Yaskawa INFORM job: BATMAN_4SPOINY2.JBI

/JOB
//NAME BATMAN_4SPOINY2
///FOLDERNAME KRIS-SCIANA
//POS
///NPOS 293,293,243,19,0,0
///TOOL 0
///POSTYPE PULSE
///PULSE
C00000=27461,19727,-15013,5964,93200,7919
C00001=53930,-34836,-43070,10546,92631,-44102
C00002=59372,-32233,-36195,10185,89087,-42536
C00003=59542,-32241,-35992,10174,88938,-42491
C00004=59542,-32142,-35265,10174,88546,-42521
C00005=59542,-32241,-35992,10174,88938,-42491
C00006=60428,-32802,-36126,10115,88624,-42213
C00007=59542,-32241,-35992,10174,88938,-42491
C00008=64039,-48991,-58660,9906,93649,-40580
C00009=69362,-49546,-56329,9460,91325,-38954
C00010=72521,-45533,-52121,9188,90441,-37947
C00011=72521,-45481,-51268,9186,89947,-37982
C00012=72521,-45533,-52121,9188,90441,-37947
C00013=73752,-44607,-51263,9079,90249,-37543
C00014=72521,-45533,-52121,9188,90441,-37947
C00015=72780,-67210,-74355,9190,92926,-37677
C00016=104760,-79002,-75488,1590,83769,10908
C00017=104760,-78316,-71792,1595,81848,10885
C00018=104951,-72146,-66630,1566,81838,10949
C00019=104951,-71977,-65827,1567,81431,10946
C00020=104951,-72146,-66630,1566,81838,10949
C00021=104585,-69689,-65175,1617,82213,10830
C00022=104951,-72146,-66630,1566,81838,10949
C00023=126930,-89810,-77004,-2546,79326,20912
C00024=126930,-86182,-66696,-2587,74851,21005
C00025=124517,-79688,-62407,-2239,75475,20152
C00026=124517,-79372,-61547,-2242,75108,20158
C00027=124517,-79688,-62407,-2239,75475,20152
C00028=123608,-77929,-61403,-2108,75735,19831
C00029=124517,-79688,-62407,-2239,75475,20152
C00030=203387,-120314,-87249,-1260,66339,1853
C00031=200667,-112422,-82916,-708,67693,857
C00032=200667,-111811,-81800,-709,67321,859
C00033=200667,-112422,-82916,-708,67693,857
C00034=202283,-108660,-81695,-1019,68894,1430
C00035=200667,-112422,-82916,-708,67693,857
C00036=197903,-118206,-84689,-161,65798,-138
C00037=190700,-136110,-79236,12987,43309,-5470
C00038=193073,-133711,-78763,11750,43893,-4292
C00039=190700,-136110,-79236,12987,43309,-5470
C00040=190700,-133577,-76218,13120,42767,-5552
C00041=190700,-136110,-79236,12987,43309,-5470
C00042=159264,-85348,-72338,26469,101848,-35770
C00043=164489,-85917,-58916,26689,92487,-35917
C00044=168310,-82776,-58110,27297,92259,-34533
C00045=169943,-81162,-57428,27533,92089,-33955
C00046=168310,-82776,-58110,27297,92259,-34533
C00047=168310,-81475,-55247,27268,91281,-34761
C00048=168310,-82776,-58110,27297,92259,-34533
C00049=174818,-166728,-104111,5010,53468,-9061
C00050=151913,-165072,-108467,9162,58894,-17426
C00051=31054,-58499,-67437,-4813,86361,7552
C00052=17460,-13489,-32841,5083,88285,-10080
C00053=18511,-10450,-28211,4896,86939,-9785
C00054=18511,-10497,-27164,4898,86273,-9811
C00055=18511,-10450,-28211,4896,86939,-9785
C00056=18072,-6386,-24997,4976,87076,-9926
C00057=18511,-10450,-28211,4896,86939,-9785
C00058=19304,-17015,-37138,4755,89006,-9443
C00059=40718,-16031,-27821,-22618,89289,5458
C00060=35897,-12993,-23126,-22071,86757,4185
C00061=35408,-10854,-21474,-22011,86705,4017
C00062=35897,-12993,-23126,-22071,86757,4185
C00063=35897,-12823,-21290,-22084,85788,4364
C00064=35897,-12993,-23126,-22071,86757,4185
C00065=31722,-22647,-27301,-21597,83426,3277
C00066=29589,-18207,-23578,-21312,82862,2603
C00067=29229,-16321,-22176,-21257,82868,2471
C00068=29589,-18207,-23578,-21312,82862,2603
C00069=29589,-17904,-21603,-21354,81873,2778
C00070=29589,-18207,-23578,-21312,82862,2603
C00071=33057,-35215,-50272,-21725,90936,2406
C00072=13245,-10427,-29720,5825,88219,-11479
C00073=13394,-4718,-22818,5800,86900,-11488
C00074=18206,-7497,-25118,4952,86573,-9901
C00075=18519,-8090,-25381,4896,86408,-9803
C00076=21911,-9763,-26755,4284,86207,-8681
C00077=21762,-10624,-27040,4312,85947,-8742
C00078=25203,-13472,-28530,-1187,84834,1033
C00079=19550,-17151,-28181,-117,82684,-851
C00080=19443,-16796,-23929,-6731,81807,11381
C00081=20023,-18123,-24279,-6835,81387,11602
C00082=21850,-21543,-25350,-7161,80456,12281
C00083=15586,-21049,-25758,415,81887,2238
C00084=14598,-19690,-25084,2340,83349,-603
C00085=17410,-32379,-43825,1943,88285,427
C00086=62758,-61083,-67514,9356,96495,3913
C00087=199419,-126821,-93595,-3849,72358,1575
C00088=215588,-96023,-77843,-5493,79414,6921
C00089=206230,-97336,-78342,-4514,78461,3733
C00090=205980,-97628,-78299,-4491,78272,3656
C00091=198784,-97250,-78233,-3683,78060,1181
C00092=198556,-98334,-78334,-3662,77556,1119
C00093=199186,-98644,-78275,-3737,77391,1339
C00094=187587,-121388,-81242,8247,57073,-3790
C00095=198009,-126022,-79257,5356,52636,78
C00096=198735,-126438,-75439,11422,52308,-7805
C00097=182087,-109335,-69935,21135,69891,-28872
C00098=173698,-101527,-65024,22396,76730,-30869
C00099=174667,-108871,-67545,21614,70616,-31488
C00100=190087,-128682,-72511,14911,50768,-12319
C00101=165785,-126013,-84565,21580,74443,-34035
C00102=65346,-79799,-84675,10403,98195,-30166
C00103=73542,-33969,-44608,8971,95126,-24746
C00104=73466,-33578,-44297,8974,95141,-24769
C00105=56512,-3179,-12316,26889,108547,-27571
C00106=55135,-19184,-25463,26231,99696,-30127
C00107=47657,-21774,-22421,25331,99126,-33105
C00108=47657,-23151,-32449,25918,104076,-32001
C00109=58332,-49897,-67983,12473,95404,-30979
C00110=76814,-87681,-77913,12459,85852,-4883
C00111=98077,-64526,-65270,10461,86864,2540
C00112=98077,-64004,-61535,10478,84867,2372
C00113=98452,-64122,-61596,10437,84795,2494
C00114=136766,-62959,-54295,-24287,84543,16325
C00115=133538,-79296,-61255,-19745,72823,18967
C00116=138375,-88192,-61332,-20789,69437,20890
C00117=138917,-90913,-61585,-20643,67750,20404
C00118=142002,-103150,-73880,-19907,68072,18980
C00119=156669,-121711,-96887,-11323,85539,21769
C00120=4467,-137969,-110669,-6539,34039,-3130
C00121=19856,121451,20000,-7167,97699,-79935
C00122=-30106,49565,32966,-7153,97659,-79929
///LIMIT ON
C00123=-48667,-96740,-85237,-4414,71954,-161170
C00124=-50087,-78703,-69642,-4046,71552,-161658
C00125=-49056,-78152,-68509,-4328,71190,-161282
C00126=-50087,-78703,-69642,-4046,71552,-161658
C00127=-51559,-77641,-68057,-3663,71053,-162163
C00128=-50087,-78703,-69642,-4046,71552,-161658
C00129=-68843,-102087,-91870,723,73949,-168126
C00130=-111940,-50657,-63992,-844,88968,-142439
C00131=-116747,-35976,-49037,-28,87281,-144022
C00132=-120801,-38775,-48909,662,85780,-145375
C00133=-120801,-38756,-47729,662,85062,-145378
C00134=-120801,-38775,-48909,662,85780,-145375
C00135=-121754,-36220,-46769,824,85785,-145694
C00136=-120801,-38775,-48909,662,85780,-145375
C00137=-125210,-26619,-58097,1431,97733,-146711
C00138=-131530,-17132,-45035,1132,94544,-146201
C00139=-131530,-17365,-44333,1131,93991,-146205
C00140=-131530,-17132,-45035,1132,94544,-146201
C00141=-132146,-15038,-43228,1237,94517,-146399
C00142=-131530,-17132,-45035,1132,94544,-146201
C00143=-161629,-2767,-38396,12559,109608,-190789
C00144=-160029,-4292,-24208,11904,100070,-191215
C00145=-160029,-4346,-23457,11882,99590,-191262
C00146=-160029,-4292,-24208,11904,100070,-191215
C00147=-159085,-3286,-23121,11882,99786,-190918
C00148=-160029,-4292,-24208,11904,100070,-191215
C00149=-164567,11803,-19941,12295,106250,-192160
C00150=-157312,-13774,-45091,-2984,98065,-146499
C00151=-206670,-20774,-45162,4390,94951,-162466
C00152=-207434,-3536,-26344,4477,92277,-162812
C00153=-207134,-1926,-24499,4435,91966,-162724
C00154=-207434,-3536,-26344,4477,92277,-162812
C00155=-208212,-2907,-24823,4582,91708,-163090
C00156=-207434,-3536,-26344,4477,92277,-162812
C00157=-203791,-18921,-42474,3974,94109,-161555
C00158=-208102,-33336,-45107,4384,70878,-171284
C00159=-208479,-26108,-38450,4536,70518,-171428
C00160=-208501,-36193,-39722,4679,66129,-171606
C00161=-213385,-11527,-27447,11970,86947,-171405
C00162=-211009,-28161,-49573,11590,91579,-170169
C00163=-152191,-54135,-82173,-578,95677,-207495
C00164=-98829,-148789,-110327,23555,60006,-190918
C00165=-63524,-94038,-77380,10109,60123,-176665
C00166=-56536,-89434,-70565,3215,56920,-170295
C00167=-56480,-89635,-70927,3185,57034,-170270
C00168=-58851,-96962,-68332,4510,51796,-171436
C00169=-51054,-86638,-67405,-5688,64202,-168107
C00170=-66960,-121145,-97778,-723,64525,-174040
C00171=-151266,-18842,-50725,13491,96086,-200286
C00172=-151199,-2206,-30574,14854,95015,-197817
C00173=-151558,-2403,-30281,14862,94131,-203931
C00174=-156353,-9182,-30957,16219,92997,-207432
C00175=-161657,-20517,-34126,16277,89446,-208209
C00176=-166380,-28855,-45761,15510,91081,-205955
C00177=-176343,-27519,-58136,14484,97680,-202423
C00178=-146432,-62330,-79152,8575,88774,-157888
C00179=-135076,-29913,-53110,6046,88415,-154204
C00180=-132700,-21303,-45243,5501,87836,-153459
C00181=-120110,-24629,-45165,-11500,84499,-143667
C00182=-116346,-38856,-49381,-12534,80425,-141997
C00183=-112747,-49987,-51295,-13579,76569,-140328
C00184=-112325,-51024,-51497,-13698,76241,-140141
C00185=-106405,-53098,-58914,-14887,80672,-138578
C00186=-95224,-20863,-45190,-12261,93737,-137947
C00187=-95224,-20863,-45190,-12261,93737,-137947
C00188=-95567,-18712,-43618,-12211,93824,-138068
C00189=2669,-23463,-43684,-12198,93814,-143081
C00190=12882,-2853,-23046,-12338,79295,-114850
C00191=140228,6881,-10027,16067,87628,-189683
C00192=178636,-26215,-18003,9541,69682,-178042
C00193=190464,-1998,2686,-1702,78410,-173449
C00194=190464,-1807,3325,-1703,78115,-173446
C00195=190464,-1851,3178,-1703,78183,-173446
C00196=190464,-572,4236,-1705,78187,-173446
C00197=190079,-3448,589,-1660,78950,-173589
C00198=170718,-8896,-1072,11364,69213,-180966
C00199=176690,18547,19438,-1102,83032,-178253
C00200=176690,18907,20631,-1103,82484,-178249
C00201=176690,18865,20492,-1103,82549,-178249
C00202=176937,20672,22196,-1113,82434,-178165
C00203=176690,18518,19335,-1103,83082,-178254
C00204=159096,10761,15360,13640,71000,-185020
C00205=163699,23839,25637,3670,75746,-182781
C00206=163699,24193,26736,3676,75252,-182795
C00207=163699,24137,26562,3674,75330,-182794
C00208=164134,25799,28176,3622,75172,-182647
C00209=163699,23793,25492,3667,75812,-182780
C00210=150784,29671,32882,15137,71440,-188000
C00211=157156,47733,49397,1195,75308,-184939
C00212=157156,48104,50383,1197,74893,-184942
C00213=157156,48016,50149,1197,74991,-184943
C00214=157735,49760,52060,1141,74703,-184746
C00215=157156,47434,48587,1193,75652,-184937
C00216=142367,63352,68521,16801,68626,-191483
C00217=154723,16721,17849,2207,78471,-185762
C00218=154723,17075,19023,2210,77929,-185773
C00219=154723,17004,18788,2210,78036,-185770
C00220=155361,18646,20317,2147,77921,-185553
C00221=154295,15409,15439,2245,79287,-185894
C00222=152548,-46037,-33001,14724,72703,-187200
C00223=173063,-35885,-19745,11040,66557,-180364
C00224=172381,-30459,-14817,12966,67685,-183662
C00225=189647,-41939,-21829,9364,63743,-177626
C00226=212432,-47441,-24871,3550,60965,-169203
C00227=222510,-46248,-24162,762,60877,-165387
C00228=221072,-55571,-31663,-1225,60729,-162686
C00229=183831,-42837,-24403,-640,62781,-163481
C00230=184368,-37494,-19337,-786,62417,-163277
C00231=169590,-25113,-11382,3214,64110,-168775
C00232=153390,312,7747,7325,66459,-174651
C00233=148403,13068,18934,8546,66622,-176472
C00234=147511,16247,21849,8770,66559,-176807
C00235=141966,-23210,-23563,9637,74772,-178174
C00236=49773,-23266,-23600,9630,74761,-174606
C00237=11499,-91272,-60439,14826,66037,-186980
C00238=24614,139305,42242,-12105,94129,-241398
C00239=23281,113263,30549,-9123,91006,-253685
C00240=55336,36118,-12147,-9115,91117,-253682
C00241=110497,-96010,-85203,-9082,91337,-253646
C00242=110132,-97701,-85894,-9078,90857,-326888
C00243=231444,-97696,-85555,14457,66885,-341831
C00244=239081,-48934,-58681,12347,86500,-340546
C00245=232436,-33273,-43061,13430,86148,-342856
C00246=232487,-32587,-41956,13424,85819,-342875
C00247=232487,-32542,-40985,13430,85259,-342937
C00248=232487,-32587,-41956,13424,85819,-342875
C00249=232629,-30129,-40306,13401,86035,-342805
C00250=232487,-32587,-41956,13424,85819,-342875
C00251=213809,-15512,-33444,15950,92576,-348489
C00252=216143,-7692,-23925,15635,90358,-347968
C00253=216143,-7698,-22988,15630,89798,-348040
C00254=216143,-7692,-23925,15635,90358,-347968
C00255=216488,-5395,-22087,15594,90340,-347850
C00256=216143,-7692,-23925,15635,90358,-347968
C00257=207069,12956,-7235,16611,92452,-350833
C00258=206195,16842,-2970,16681,92025,-351195
C00259=206195,16846,-1900,16669,91395,-351281
C00260=206195,16842,-2970,16681,92025,-351195
C00261=206613,19062,-907,16640,91818,-351079
C00262=206195,16842,-2970,16681,92025,-351195
C00263=210833,19416,-576,16221,90958,-349729
C00264=209935,25164,4669,16310,90872,-350053
C00265=209935,25181,5707,16303,90266,-350133
C00266=209935,25164,4669,16310,90872,-350053
C00267=210302,27507,6947,16270,90609,-349961
C00268=209935,25164,4669,16310,90872,-350053
C00269=202776,46738,24588,16950,91193,-352506
C00270=202171,51343,31379,16979,89579,-352941
C00271=202171,51457,32428,16976,89018,-353018
C00272=202171,51343,31379,16979,89579,-352941
C00273=202544,53678,33951,16947,89134,-352871
C00274=202171,51343,31379,16979,89579,-352941
C00275=210768,8740,-16259,16329,94978,-349219
C00276=216926,676,-19392,15562,91669,-347534
C00277=220414,8220,-10388,13170,90389,-353505
C00278=232512,-10946,-26241,11631,88471,-349576
C00279=227494,-25690,-36969,12302,88249,-351307
C00280=237440,-37130,-44669,10939,85718,-348148
C00281=231683,-43662,-56537,11755,90384,-349677
C00282=231683,-43662,-56537,11755,90384,-349677
C00283=240298,-51036,-57572,3930,82785,-334851
C00284=225025,-34742,-47804,6828,86146,-339832
C00285=212279,-13510,-33247,9067,89308,-343887
C00286=207270,-2378,-24690,9890,90330,-345482
C00287=206374,470,-22476,10033,90539,-345765
C00288=201120,-19837,-47084,10933,95828,-347061
C00289=121938,-115164,-95780,1417,89212,-367207
C00290=62315,-114908,-95780,1418,89212,-367206
C00291=62316,-114908,-95779,1418,89212,-367205
C00292=29956,140088,42679,-12136,94183,-404796
///LIMIT OFF
BC00000=80599,337603,478005
BC00001=163893,318206,473102
BC00002=163893,318206,473102
BC00003=163893,318206,473102
BC00004=163893,318206,473102
BC00005=163893,318206,473102
BC00006=163893,318206,473102
BC00007=163893,318206,473102
BC00008=163893,318206,473102
BC00009=163893,318206,473102
BC00010=163893,318206,473102
BC00011=163893,318206,473102
BC00012=163893,318206,473102
BC00013=163893,318206,473102
BC00014=163893,318206,473102
BC00015=163893,318206,473102
BC00016=163893,318206,473102
BC00017=163893,318206,473102
BC00018=163893,318206,473102
BC00019=163893,318206,473102
BC00020=163893,318206,473102
BC00021=163893,318206,473102
BC00022=163893,318206,473102
BC00023=163893,318206,473102
BC00024=163893,318206,473102
BC00025=163893,318206,473102
BC00026=163893,318206,473102
BC00027=163893,318206,473102
BC00028=163893,318206,473102
BC00029=163893,318206,473102
BC00030=163893,318206,473102
BC00031=163893,318206,473102
BC00032=163893,318206,473102
BC00033=163893,318206,473102
BC00034=163893,318206,473102
BC00035=163893,318206,473102
BC00036=163893,318206,473102
BC00037=163893,318206,473102
BC00038=163893,318206,473102
BC00039=163893,318206,473102
BC00040=163893,318206,473102
BC00041=163893,318206,473102
BC00042=163892,318206,473100
BC00043=163892,318207,473095
BC00044=163892,318207,473095
BC00045=163892,318207,473095
BC00046=163892,318207,473095
BC00047=163892,318207,473095
BC00048=163892,318207,473095
BC00049=163893,318206,473102
BC00050=163893,318206,473102
BC00051=163893,318206,473102
BC00052=163893,318206,473102
BC00053=163893,318206,473102
BC00054=163893,318206,473102
BC00055=163893,318206,473102
BC00056=163893,318206,473102
BC00057=163893,318206,473102
BC00058=163893,318206,473102
BC00059=163893,318206,473102
BC00060=163893,318206,473102
BC00061=163893,318206,473102
BC00062=163893,318206,473102
BC00063=163893,318206,473102
BC00064=163893,318206,473102
BC00065=163893,318206,473102
BC00066=163893,318206,473102
BC00067=163893,318206,473102
BC00068=163893,318206,473102
BC00069=163893,318206,473102
BC00070=163893,318206,473102
BC00071=163893,318206,473102
BC00072=163893,318206,473102
BC00073=163893,318206,473102
BC00074=163893,318206,473102
BC00075=163893,318206,473102
BC00076=163893,318206,473102
BC00077=163893,318206,473102
BC00078=163893,318206,473102
BC00079=163893,318206,473102
BC00080=163893,318206,473102
BC00081=163893,318206,473102
BC00082=163893,318206,473102
BC00083=163894,318206,473105
BC00084=163894,318206,473105
BC00085=163894,318206,473105
BC00086=163894,318207,608827
BC00087=163894,318207,473102
BC00088=163894,318207,473102
BC00089=163894,318207,473102
BC00090=163894,318207,473102
BC00091=163894,318207,473102
BC00092=163894,318207,473102
BC00093=163894,318207,473102
BC00094=163894,318207,473102
BC00095=163894,318207,473102
BC00096=163894,318207,473102
BC00097=163894,318207,473102
BC00098=163894,318207,473102
BC00099=163894,318207,473102
BC00100=163894,318207,473102
BC00101=163894,318207,473102
BC00102=163894,318207,473102
BC00103=163894,318207,473102
BC00104=163894,318207,473102
BC00105=163894,318207,473102
BC00106=163894,318207,473102
BC00107=163894,318207,473102
BC00108=163894,318207,473102
BC00109=163894,318207,473102
BC00110=163894,318207,473102
BC00111=163894,318207,473102
BC00112=163894,318207,473102
BC00113=163894,318207,473102
BC00114=163894,318207,473102
BC00115=163894,318207,473102
BC00116=163894,318207,473102
BC00117=163894,318207,473102
BC00118=163894,318207,473102
BC00119=163894,318207,706181
BC00120=112319,5379,1050005
BC00121=125260,5957,1075157
BC00122=125260,5957,1075157
BC00123=255263,5047,617472
BC00124=255263,5047,617472
BC00125=255263,5047,617472
BC00126=255263,5047,617472
BC00127=255263,5047,617472
BC00128=255263,5047,617472
BC00129=255263,5047,617472
BC00130=255263,5047,617472
BC00131=255263,5047,617472
BC00132=255263,5047,617472
BC00133=255263,5047,617472
BC00134=255263,5047,617472
BC00135=255263,5047,617472
BC00136=255263,5047,617472
BC00137=255263,5047,617472
BC00138=255263,5047,617472
BC00139=255263,5047,617472
BC00140=255263,5047,617472
BC00141=255263,5047,617472
BC00142=255263,5047,617472
BC00143=255263,5047,617472
BC00144=255263,5047,617472
BC00145=255263,5047,617472
BC00146=255263,5047,617472
BC00147=255263,5047,617472
BC00148=255263,5047,617472
BC00149=255263,5047,617472
BC00150=255263,5047,617472
BC00151=255263,5047,617472
BC00152=255263,5047,617472
BC00153=255262,5048,617469
BC00154=255263,5047,617472
BC00155=255263,5047,617472
BC00156=255263,5047,617472
BC00157=255263,5047,617472
BC00158=255263,5047,617472
BC00159=255263,5047,617472
BC00160=255263,5047,617472
BC00161=255263,5047,617472
BC00162=255263,5047,617472
BC00163=255262,5047,617469
BC00164=255262,5047,617469
BC00165=255262,5047,617469
BC00166=255262,5047,617469
BC00167=255261,5048,617462
BC00168=255261,5048,617462
BC00169=255261,5048,617462
BC00170=255261,5048,617462
BC00171=255261,5048,617462
BC00172=255261,5048,617460
BC00173=255261,5048,617460
BC00174=255261,5048,617460
BC00175=255261,5048,617460
BC00176=255261,5048,617460
BC00177=255261,5048,617460
BC00178=255261,5048,617460
BC00179=255262,5048,617458
BC00180=255262,5048,617458
BC00181=255262,5048,617458
BC00182=255262,5048,617458
BC00183=255262,5048,617458
BC00184=255262,5048,617458
BC00185=255262,5048,617458
BC00186=255262,5048,1054021
BC00187=364357,5048,1054021
BC00188=346085,493744,1054021
BC00189=119927,493744,1054021
BC00190=122126,493982,1062735
BC00191=316085,494322,354264
BC00192=316085,376158,354264
BC00193=316085,376158,354264
BC00194=316085,376158,354264
BC00195=316085,376158,354264
BC00196=316085,376158,354264
BC00197=316085,376158,354264
BC00198=316085,376158,354264
BC00199=316085,376158,354264
BC00200=316085,376158,354264
BC00201=316085,376158,354264
BC00202=316085,376158,354264
BC00203=316085,376158,354264
BC00204=316085,376158,354264
BC00205=316085,376158,354264
BC00206=316085,376158,354264
BC00207=316085,376158,354264
BC00208=316085,376158,354264
BC00209=316085,376158,354264
BC00210=316085,376158,354264
BC00211=316085,376158,354264
BC00212=316085,376158,354264
BC00213=316085,376158,354264
BC00214=316085,376158,354264
BC00215=316085,376158,354264
BC00216=316085,376158,354264
BC00217=316085,310375,354264
BC00218=316085,310375,354264
BC00219=316085,310375,354264
BC00220=316085,310375,354264
BC00221=316085,310375,354264
BC00222=316085,310375,354264
BC00223=316085,310375,354264
BC00224=316083,310375,354262
BC00225=316083,310375,354262
BC00226=316083,310375,354262
BC00227=316083,310375,354262
BC00228=316083,310375,354262
BC00229=316083,310375,354262
BC00230=316083,310375,354262
BC00231=316083,310375,354262
BC00232=316083,310375,354262
BC00233=316083,310375,354262
BC00234=316083,310375,354262
BC00235=316083,310374,354261
BC00236=221693,504700,545055
BC00237=139211,579237,982811
BC00238=124231,580310,1074882
BC00239=85429,579747,1064499
BC00240=244755,514688,1010883
BC00241=393595,402951,918797
BC00242=393595,99043,918797
BC00243=393595,99043,199678
BC00244=398179,136533,199678
BC00245=398179,136533,199674
BC00246=398179,136533,199674
BC00247=398179,136533,199674
BC00248=398179,136533,199674
BC00249=398179,136533,199674
BC00250=398179,136533,199674
BC00251=398179,136533,199674
BC00252=398179,136532,199672
BC00253=398179,136532,199672
BC00254=398179,136532,199672
BC00255=398179,136532,199672
BC00256=398179,136532,199672
BC00257=398179,136532,199672
BC00258=398179,136532,199672
BC00259=398179,136532,199672
BC00260=398179,136532,199672
BC00261=398179,136532,199672
BC00262=398179,136532,199672
BC00263=398179,99664,199672
BC00264=398179,99664,199672
BC00265=398179,99664,199672
BC00266=398179,99664,199672
BC00267=398179,99664,199672
BC00268=398179,99664,199672
BC00269=398179,99664,199672
BC00270=398179,99664,199672
BC00271=398179,99664,199672
BC00272=398179,99664,199672
BC00273=398179,99664,199672
BC00274=398179,99664,199672
BC00275=398179,99664,199672
BC00276=398179,99664,199672
BC00277=398179,99664,199672
BC00278=398179,99664,199672
BC00279=398179,149360,199672
BC00280=398179,149360,199672
BC00281=398179,149360,199672
BC00282=351196,62906,171676
BC00283=351196,62906,171676
BC00284=351196,62906,171676
BC00285=351196,62906,171676
BC00286=351196,62906,171676
BC00287=351196,62906,171676
BC00288=351196,62906,171676
BC00289=397107,62906,780423
BC00290=397107,492277,780423
BC00291=397107,492277,780421
BC00292=68537,642032,1075143
EC00000=-811452,-554689
EC00001=-811450,-554689
EC00002=-811450,-554689
EC00003=-811450,-554689
EC00004=-811450,-554689
EC00005=-811450,-554689
EC00006=-811450,-554689
EC00007=-811450,-554689
EC00008=-811450,-554689
EC00009=-811450,-554689
EC00010=-811450,-554689
EC00011=-811450,-554689
EC00012=-811450,-554689
EC00013=-811450,-554689
EC00014=-811450,-554689
EC00015=-811450,-554689
EC00016=-811450,-554689
EC00017=-811450,-554689
EC00018=-811450,-554689
EC00019=-811450,-554689
EC00020=-811450,-554689
EC00021=-811450,-554689
EC00022=-811450,-554689
EC00023=-811450,-554689
EC00024=-811450,-554689
EC00025=-811450,-554689
EC00026=-811450,-554689
EC00027=-811450,-554689
EC00028=-811450,-554689
EC00029=-811450,-554689
EC00030=-811447,-554690
EC00031=-811443,-554690
EC00032=-811443,-554690
EC00033=-811443,-554690
EC00034=-811443,-554690
EC00035=-811450,-554689
EC00036=-811450,-554689
EC00037=-811450,-554689
EC00038=-811450,-554689
EC00039=-811450,-554689
EC00040=-811450,-554689
EC00041=-811450,-554689
EC00042=-811450,-554689
EC00043=-811450,-554689
EC00044=-811450,-554689
EC00045=-811450,-554689
EC00046=-811450,-554689
EC00047=-811450,-554689
EC00048=-811450,-554689
EC00049=-811450,-554689
EC00050=-811450,-554689
EC00051=-811450,-554689
EC00052=-811450,-554689
EC00053=-811450,-554689
EC00054=-811450,-554689
EC00055=-811450,-554689
EC00056=-811450,-554689
EC00057=-811450,-554689
EC00058=-811450,-554689
EC00059=-811450,-554689
EC00060=-811450,-554689
EC00061=-811450,-554689
EC00062=-811450,-554689
EC00063=-811452,-554689
EC00064=-811452,-554689
EC00065=-811452,-554689
EC00066=-811451,-554689
EC00067=-811451,-554689
EC00068=-811451,-554689
EC00069=-811451,-554689
EC00070=-811451,-554689
EC00071=-811451,-554689
EC00072=-811451,-554689
EC00073=-811451,-554689
EC00074=-811451,-554689
EC00075=-811451,-554689
EC00076=-811451,-554689
EC00077=-811451,-554689
EC00078=-811451,-554689
EC00079=-811451,-554689
EC00080=-811451,-554689
EC00081=-811451,-554689
EC00082=-811451,-554689
EC00083=-811451,-554689
EC00084=-811451,-554689
EC00085=-811451,-554689
EC00086=-811451,-554689
EC00087=-811451,-554689
EC00088=-811451,-554689
EC00089=-811451,-554689
EC00090=-811451,-554689
EC00091=-811451,-554689
EC00092=-811451,-554689
EC00093=-811451,-554689
EC00094=-811451,-554689
EC00095=-811451,-554689
EC00096=-811451,-554689
EC00097=-811451,-554689
EC00098=-811451,-554689
EC00099=-811451,-554689
EC00100=-363208,-550746
EC00101=-363208,-550746
EC00102=-363208,-550746
EC00103=-363208,-550746
EC00104=-363208,-550746
EC00105=-363208,-550746
EC00106=-363208,-550746
EC00107=-363208,-550746
EC00108=-363208,-550746
EC00109=-363208,-550746
EC00110=-363208,-550746
EC00111=-363208,-550746
EC00112=-363208,-550746
EC00113=-363208,-550746
EC00114=-363208,-550746
EC00115=-363208,-550746
EC00116=-363208,-550746
EC00117=-363208,-550746
EC00118=-363208,-550746
EC00119=-363208,-550746
EC00120=-363208,-550746
EC00121=-363208,-550746
EC00122=-363208,-550746
EC00123=-363208,-550746
EC00124=-363208,-550746
EC00125=-363208,-550746
EC00126=-363208,-550746
EC00127=-363208,-550746
EC00128=-363208,-550746
EC00129=-363208,-550746
EC00130=-363208,-550746
EC00131=-363208,-550746
EC00132=-363208,-550746
EC00133=-363208,-550746
EC00134=-363208,-550746
EC00135=-363208,-550746
EC00136=-363208,-550746
EC00137=-363207,-550746
EC00138=-363207,-550746
EC00139=-363207,-550746
EC00140=-363207,-550746
EC00141=-363207,-550746
EC00142=-363206,-550746
EC00143=-363206,-550746
EC00144=-363206,-550746
EC00145=-363206,-550746
EC00146=-363206,-550746
EC00147=-363206,-550746
EC00148=-363206,-550746
EC00149=-363206,-550746
EC00150=-363206,-550746
EC00151=-363206,-550746
EC00152=-363206,-550746
EC00153=-363206,-550746
EC00154=-363206,-550746
EC00155=-363206,-550746
EC00156=-363206,-550746
EC00157=-363206,-550746
EC00158=0,0
EC00159=-802750,0
EC00160=-802750,0
EC00161=-802750,0
EC00162=-802750,0
EC00163=-802750,0
EC00164=-802750,0
EC00165=-802750,0
EC00166=-802750,0
EC00167=-802750,0
EC00168=-802750,0
EC00169=-802750,0
EC00170=-802750,0
EC00171=-802750,0
EC00172=-802750,0
EC00173=-802750,0
EC00174=-802750,0
EC00175=-802750,0
EC00176=-802750,0
EC00177=-802750,0
EC00178=-802750,0
EC00179=-802750,0
EC00180=-802750,0
EC00181=-802750,0
EC00182=-802750,0
EC00183=-802750,0
EC00184=-802749,0
EC00185=-802749,0
EC00186=-802749,0
EC00187=-802749,0
EC00188=-802749,0
EC00189=-802749,0
EC00190=-802749,0
EC00191=-802749,0
EC00192=-802749,0
EC00193=-802749,0
EC00194=-802749,0
EC00195=-802748,0
EC00196=-802748,0
EC00197=793507,0
EC00198=793506,-1
EC00199=793506,-1
EC00200=793506,-1
EC00201=793506,-1
EC00202=793506,-1
EC00203=793506,-1
EC00204=793506,-1
EC00205=793505,-1
EC00206=793505,-1
EC00207=793505,-1
EC00208=793505,-1
EC00209=793505,-1
EC00210=793504,-1
EC00211=793504,-1
EC00212=793504,-1
EC00213=793504,-1
EC00214=793504,-1
EC00215=793504,-1
EC00216=793504,-1
EC00217=793504,-1
EC00218=793504,-1
EC00219=793504,-1
EC00220=793504,-1
EC00221=793504,-1
EC00222=793504,-1
EC00223=793504,-1
EC00224=793504,-1
EC00225=793504,-1
EC00226=793504,-1
EC00227=793504,-1
EC00228=793504,-1
EC00229=793504,-1
EC00230=793504,-1
EC00231=793504,-1
EC00232=793504,-1
EC00233=793504,-1
EC00234=793504,-1
EC00235=793504,-1
EC00236=793504,-1
EC00237=793504,-1
EC00238=793504,-1
EC00239=793504,-1
EC00240=793504,-1
EC00241=793503,548424
EC00242=0,-1
///POSTYPE BASE
///RECTAN
///RCONF 0,0,0,0,1,0,0,0,0,0,0,0,0,0,0,0,0,0,0,0,0,0,0,0
P00006=2.006,1.622,-0.565,0.0000,0.0000,0.0000
P00021=0.073,2.058,-0.109,0.0000,0.0000,0.0000
P00022=2.006,1.622,-0.565,0.0000,0.0000,0.0000
///RCONF 0,0,0,0,0,0,0,0,0,0,0,0,0,0,0,0,0,0,0,0,0,0,0,0
P00023=-2.957,-4.083,2.762,0.0000,0.0000,0.0000
P00024=-1.466,-0.226,-0.419,0.0000,0.0000,0.0000
P00025=3.643,0.007,-2.585,0.0000,0.0000,0.0000
P00026=2.644,0.055,-2.583,0.0000,0.0000,0.0000
P00027=2.278,0.099,-4.210,0.0000,0.0000,0.0000
P00028=-1.778,-0.182,-2.050,0.0000,0.0000,0.0000
P00029=1.749,4.006,-0.261,0.0000,0.0000,0.0000
P00030=-0.014,-0.768,0.131,0.0000,0.0000,0.0000
///RCONF 0,0,0,0,1,0,0,0,0,0,0,0,0,0,0,0,0,0,0,0,0,0,0,0
P00034=-8.151,9.743,-4.393,0.0000,0.0000,0.0000
///RCONF 0,0,0,0,0,0,0,0,0,0,0,0,0,0,0,0,0,0,0,0,0,0,0,0
P00035=0.390,-0.027,1.040,0.0000,0.0000,0.0000
P00036=-2.434,0.084,0.197,0.0000,0.0000,0.0000
P00037=-1.075,5.090,-3.949,0.0000,0.0000,0.0000
P00040=2.716,-0.016,3.014,0.0000,0.0000,0.0000
P00041=-0.109,0.014,0.966,0.0000,0.0000,0.0000
P00042=-0.220,0.371,-0.613,0.0000,0.0000,0.0000
P00043=-0.179,-5.890,-3.227,0.0000,0.0000,0.0000
//INST
///DATE 2024/07/30 17:33
///ATTR SC,RW
///GROUP1 RB1,BS1
///GROUP2 ST1
NOP
SFTOF
MOVJ C00000 BC00000 VJ=100.00  +MOVJ EC00000 VJ=100.00
'SZUKANIE
SFTOF
MOVJ C00001 BC00001 VJ=100.00  +MOVJ EC00001 VJ=30.00
MOVL C00002 BC00002 V=83.3  +MOVJ EC00002 VJ=15.00
MOVL C00003 BC00003 V=83.3  +MOVJ EC00003 VJ=15.00
REFP 3 RB1 C00004 BC00004
CALL JOB:SEARCH-R1
SET P026 P006
SFTON P026
MOVL C00005 BC00005 V=83.3  +MOVJ EC00004 VJ=15.00
REFP 3 RB1 C00006 BC00006
CALL JOB:SEARCH-R1
SET P026 P006
MOVL C00007 BC00007 V=83.3  +MOVJ EC00005 VJ=15.00
SFTOF
MOVL C00008 BC00008 V=83.3  +MOVJ EC00006 VJ=15.00
MOVL C00009 BC00009 V=83.3  +MOVJ EC00007 VJ=15.00
MOVL C00010 BC00010 V=83.3  +MOVJ EC00008 VJ=15.00
REFP 3 RB1 C00011 BC00011
CALL JOB:SEARCH-R1
SET P027 P006
SFTON P027
MOVL C00012 BC00012 V=83.3  +MOVJ EC00009 VJ=15.00
REFP 3 RB1 C00013 BC00013
CALL JOB:SEARCH-R1
SET P027 P006
MOVL C00014 BC00014 V=83.3  +MOVJ EC00010 VJ=15.00
SFTOF
MOVJ C00015 BC00015 VJ=100.00  +MOVJ EC00011 VJ=100.00
SFTOF
MOVJ C00016 BC00016 VJ=100.00  +MOVJ EC00012 VJ=100.00
MOVL C00017 BC00017 V=83.3  +MOVJ EC00013 VJ=15.00
MOVL C00018 BC00018 V=83.3  +MOVJ EC00014 VJ=15.00
REFP 3 RB1 C00019 BC00019
CALL JOB:SEARCH-R1
SET P029 P006
SFTON P029
MOVL C00020 BC00020 V=83.3  +MOVJ EC00015 VJ=15.00
REFP 3 RB1 C00021 BC00021
CALL JOB:SEARCH-R1
SET P029 P006
MOVL C00022 BC00022 V=83.3  +MOVJ EC00016 VJ=15.00
SFTOF
MOVL C00023 BC00023 V=83.3  +MOVJ EC00017 VJ=15.00
MOVL C00024 BC00024 V=83.3  +MOVJ EC00018 VJ=15.00
MOVL C00025 BC00025 V=83.3  +MOVJ EC00019 VJ=15.00
REFP 3 RB1 C00026 BC00026
CALL JOB:SEARCH-R1
SET P030 P006
SFTON P030
MOVL C00027 BC00027 V=83.3  +MOVJ EC00020 VJ=15.00
REFP 3 RB1 C00028 BC00028
CALL JOB:SEARCH-R1
SET P030 P006
MOVL C00029 BC00029 V=83.3  +MOVJ EC00021 VJ=15.00
SFTOF
MOVL C00030 BC00030 V=250.0  +MOVJ EC00022 VJ=15.00
MOVL C00031 BC00031 V=83.3  +MOVJ EC00023 VJ=15.00
REFP 3 RB1 C00032 BC00032
CALL JOB:SEARCH-R1
SET P036 P006
SFTON P036
MOVL C00033 BC00033 V=83.3  +MOVJ EC00024 VJ=15.00
REFP 3 RB1 C00034 BC00034
CALL JOB:SEARCH-R1
SET P036 P006
MOVL C00035 BC00035 V=83.3  +MOVJ EC00025 VJ=15.00
SFTOF
MOVL C00036 BC00036 V=11.0  +MOVJ EC00026 VJ=0.78
MOVL C00037 BC00037 V=83.3  +MOVJ EC00027 VJ=15.00
REFP 3 RB1 C00038 BC00038
CALL JOB:SEARCH-R1
SET P040 P006
SFTON P040
MOVL C00039 BC00039 V=83.3  +MOVJ EC00028 VJ=15.00
REFP 3 RB1 C00040 BC00040
CALL JOB:SEARCH-R1
SET P040 P006
MOVL C00041 BC00041 V=83.3  +MOVJ EC00029 VJ=15.00
SFTOF
MOVJ C00042 BC00042 VJ=100.00  +MOVJ EC00030 VJ=0.78
MOVJ C00043 BC00043 VJ=100.00  +MOVJ EC00031 VJ=100.00
MOVL C00044 BC00044 V=83.3  +MOVJ EC00032 VJ=15.00
REFP 3 RB1 C00045 BC00045
CALL JOB:SEARCH-R1
SET P041 P006
SFTON P041
MOVL C00046 BC00046 V=83.3  +MOVJ EC00033 VJ=15.00
REFP 3 RB1 C00047 BC00047
CALL JOB:SEARCH-R1
SET P041 P006
MOVL C00048 BC00048 V=83.3  +MOVJ EC00034 VJ=15.00
SFTOF
MOVL C00049 BC00049 V=250.0  +MOVJ EC00035 VJ=15.00
MOVJ C00050 BC00050 VJ=100.00  +MOVJ EC00036 VJ=15.00
MOVJ C00051 BC00051 VJ=100.00  +MOVJ EC00037 VJ=100.00
MOVJ C00052 BC00052 VJ=100.00  +MOVJ EC00038 VJ=100.00
MOVL C00053 BC00053 V=83.3  +MOVJ EC00039 VJ=15.00
REFP 3 RB1 C00054 BC00054
CALL JOB:SEARCH-R1
SET P037 P006
SFTON P037
MOVL C00055 BC00055 V=83.3  +MOVJ EC00040 VJ=15.00
REFP 3 RB1 C00056 BC00056
CALL JOB:SEARCH-R1
SET P037 P006
MOVL C00057 BC00057 V=83.3  +MOVJ EC00041 VJ=15.00
MOVJ C00058 BC00058 VJ=100.00  +MOVJ EC00042 VJ=100.00
MOVJ C00059 BC00059 VJ=100.00  +MOVJ EC00043 VJ=100.00
MOVL C00060 BC00060 V=83.3  +MOVJ EC00044 VJ=15.00
REFP 3 RB1 C00061 BC00061
CALL JOB:SEARCH-R1
SET P042 P006
SFTOF
SFTON P042
MOVL C00062 BC00062 V=83.3  +MOVJ EC00045 VJ=15.00
REFP 3 RB1 C00063 BC00063
CALL JOB:SEARCH-R1
SET P042 P006
MOVL C00064 BC00064 V=83.3  +MOVJ EC00046 VJ=15.00
SFTOF
MOVJ C00065 BC00065 VJ=100.00  +MOVJ EC00047 VJ=100.00
MOVL C00066 BC00066 V=83.3  +MOVJ EC00048 VJ=15.00
REFP 3 RB1 C00067 BC00067
CALL JOB:SEARCH-R1
SET P042 P006
SFTON P042
MOVL C00068 BC00068 V=83.3  +MOVJ EC00049 VJ=15.00
REFP 3 RB1 C00069 BC00069
CALL JOB:SEARCH-R1
SET P042 P006
MOVL C00070 BC00070 V=83.3  +MOVJ EC00050 VJ=15.00
SFTOF
MOVJ C00071 BC00071 VJ=100.00  +MOVJ EC00051 VJ=100.00
SFTOF
MOVL C00072 BC00072 V=166.7  +MOVJ EC00052 VJ=15.00
SFTON P037
MACRO1 MJ#(0) ARGF7
MOVL C00073 BC00073 V=83.3  +MOVJ EC00053 VJ=100.00
ARCON
MOVL C00074 BC00074 V=10.0  +MOVJ EC00054 VJ=100.00
MOVL C00075 BC00075 V=10.0  +MOVJ EC00055 VJ=100.00
MOVL C00076 BC00076 V=10.0  +MOVJ EC00056 VJ=100.00
MOVL C00077 BC00077 V=10.0  +MOVJ EC00057 VJ=100.00
MOVL C00078 BC00078 V=10.0  +MOVJ EC00058 VJ=100.00
SFTOF
SFTON P042
MOVL C00079 BC00079 V=10.0  +MOVJ EC00059 VJ=100.00
SFTOF
SFTON P043
MOVL C00080 BC00080 V=10.0  +MOVJ EC00060 VJ=100.00
MACRO1 MJ#(0) ARGF7
MOVL C00081 BC00081 V=10.0  +MOVJ EC00061 VJ=100.00
MOVL C00082 BC00082 V=10.0  +MOVJ EC00062 VJ=100.00
MOVL C00083 BC00083 V=10.0  +MOVJ EC00063 VJ=100.00
MOVL C00084 BC00084 V=10.0  +MOVJ EC00064 VJ=20.00
ARCOF
MOVJ C00085 BC00085 VJ=20.00  +MOVJ EC00065 VJ=20.00
SFTOF
MOVJ C00086 BC00086 VJ=100.00  +MOVJ EC00066 VJ=20.00
MOVJ C00087 BC00087 VJ=100.00  +MOVJ EC00067 VJ=20.00
SFTON P036
MOVJ C00088 BC00088 VJ=20.00  +MOVJ EC00068 VJ=100.00
ARCON
MOVL C00089 BC00089 V=10.0  +MOVJ EC00069 VJ=20.00
TIMER T=0.10
MOVL C00090 BC00090 V=8.3  +MOVJ EC00070 VJ=20.00
MOVL C00091 BC00091 V=8.3  +MOVJ EC00071 VJ=20.00
MOVL C00092 BC00092 V=10.0  +MOVJ EC00072 VJ=20.00
MOVL C00093 BC00093 V=10.0  +MOVJ EC00073 VJ=20.00
MOVL C00094 BC00094 V=10.0  +MOVJ EC00074 VJ=20.00
SFTOF
SFTON P040
MOVL C00095 BC00095 V=10.0  +MOVJ EC00075 VJ=20.00
MOVL C00096 BC00096 V=10.0  +MOVJ EC00076 VJ=20.00
SFTOF
SFTON P041
MOVL C00097 BC00097 V=10.0  +MOVJ EC00077 VJ=20.00
ARCON
MOVL C00098 BC00098 V=10.0  +MOVJ EC00078 VJ=20.00
MOVL C00099 BC00099 V=10.0  +MOVJ EC00079 VJ=50.00
MOVL C00100 BC00100 V=10.0  +MOVJ EC00080 VJ=15.00
ARCOF
MOVJ C00101 BC00101 VJ=15.00  +MOVJ EC00081 VJ=15.00
SFTOF
MOVJ C00102 BC00102 VJ=30.00  +MOVJ EC00082 VJ=30.00
SFTON P027
MOVJ C00103 BC00103 VJ=30.00  +MOVJ EC00083 VJ=30.00
ARCON
MOVL C00104 BC00104 V=10.0  +MOVJ EC00084 VJ=100.00
MOVL C00105 BC00105 V=10.0  +MOVJ EC00085 VJ=20.00
SFTOF
SFTON P026
MOVL C00106 BC00106 V=10.0  +MOVJ EC00086 VJ=20.00
MOVL C00107 BC00107 V=10.0  +MOVJ EC00087 VJ=20.00
ARCOF
SFTOF
MOVJ C00108 BC00108 VJ=100.00  +MOVJ EC00088 VJ=20.00
MOVJ C00109 BC00109 VJ=30.00  +MOVJ EC00089 VJ=30.00
MOVJ C00110 BC00110 VJ=100.00  +MOVJ EC00090 VJ=20.00
MOVJ C00111 BC00111 VJ=30.00  +MOVJ EC00091 VJ=30.00
SFTON P029
MOVJ C00112 BC00112 VJ=30.00  +MOVJ EC00092 VJ=30.00
ARCON
MOVL C00113 BC00113 V=10.0  +MOVJ EC00093 VJ=20.00
MOVL C00114 BC00114 V=10.0  +MOVJ EC00094 VJ=20.00
SFTOF
SFTON P030
MOVL C00115 BC00115 V=10.0  +MOVJ EC00095 VJ=20.00
MOVL C00116 BC00116 V=10.0  +MOVJ EC00096 VJ=20.00
MOVL C00117 BC00117 V=10.0  +MOVJ EC00097 VJ=20.00
ARCOF
MOVJ C00118 BC00118 VJ=20.00  +MOVJ EC00098 VJ=20.00
SFTOF
MOVJ C00119 BC00119 VJ=100.00  +MOVJ EC00099 VJ=100.00
MOVJ C00120 BC00120 VJ=100.00  +MOVJ EC00100 VJ=100.00
CALL JOB:CLEAN-R1_LONG
MOVJ C00121 BC00121 VJ=100.00  +MOVJ EC00101 VJ=100.00
MOVJ C00122 BC00122 VJ=100.00  +MOVJ EC00102 VJ=100.00
'SZUKANIE DRUGA STRONA
MOVJ C00123 BC00123 VJ=30.00  +MOVJ EC00103 VJ=15.00
SFTOF
MOVL C00124 BC00124 V=83.3  +MOVJ EC00104 VJ=15.00
REFP 3 RB1 C00125 BC00125
CALL JOB:SEARCH-R1
SET P035 P006
SFTON P035
MOVL C00126 BC00126 V=83.3  +MOVJ EC00105 VJ=15.00
REFP 3 RB1 C00127 BC00127
CALL JOB:SEARCH-R1
SET P035 P006
MOVL C00128 BC00128 V=83.3  +MOVJ EC00106 VJ=15.00
SFTOF
MOVJ C00129 BC00129 VJ=50.00  +MOVJ EC00107 VJ=50.00
MOVJ C00130 BC00130 VJ=15.00  +MOVJ EC00108 VJ=15.00
MOVL C00131 BC00131 V=83.3  +MOVJ EC00109 VJ=15.00
MOVL C00132 BC00132 V=83.3  +MOVJ EC00110 VJ=15.00
REFP 3 RB1 C00133 BC00133
CALL JOB:SEARCH-R1
SET P026 P006
SFTON P026
MOVL C00134 BC00134 V=83.3  +MOVJ EC00111 VJ=15.00
REFP 3 RB1 C00135 BC00135
CALL JOB:SEARCH-R1
SET P026 P006
MOVL C00136 BC00136 V=83.3  +MOVJ EC00112 VJ=15.00
SFTOF
MOVL C00137 BC00137 V=83.3  +MOVJ EC00113 VJ=15.00
MOVL C00138 BC00138 V=83.3  +MOVJ EC00114 VJ=15.00
REFP 3 RB1 C00139 BC00139
CALL JOB:SEARCH-R1
SET P027 P006
SFTON P027
MOVL C00140 BC00140 V=83.3  +MOVJ EC00115 VJ=15.00
REFP 3 RB1 C00141 BC00141
CALL JOB:SEARCH-R1
SET P027 P006
MOVL C00142 BC00142 V=83.3  +MOVJ EC00116 VJ=15.00
SFTOF
MOVL C00143 BC00143 V=83.3  +MOVJ EC00117 VJ=15.00
MOVL C00144 BC00144 V=83.3  +MOVJ EC00118 VJ=15.00
REFP 3 RB1 C00145 BC00145
CALL JOB:SEARCH-R1
SET P028 P006
SFTON P028
MOVL C00146 BC00146 V=83.3  +MOVJ EC00119 VJ=15.00
REFP 3 RB1 C00147 BC00147
CALL JOB:SEARCH-R1
SET P028 P006
MOVL C00148 BC00148 V=83.3  +MOVJ EC00120 VJ=15.00
SFTOF
MOVJ C00149 BC00149 VJ=15.00  +MOVJ EC00121 VJ=15.00
MOVJ C00150 BC00150 VJ=15.00  +MOVJ EC00122 VJ=15.00
SFTOF
MOVJ C00151 BC00151 VJ=15.00  +MOVJ EC00123 VJ=15.00
MOVL C00152 BC00152 V=83.3  +MOVJ EC00124 VJ=15.00
REFP 3 RB1 C00153 BC00153
CALL JOB:SEARCH-R1
SET P034 P006
SFTON P034
MOVL C00154 BC00154 V=83.3  +MOVJ EC00125 VJ=15.00
REFP 3 RB1 C00155 BC00155
CALL JOB:SEARCH-R1
SET P034 P006
MOVL C00156 BC00156 V=83.3  +MOVJ EC00126 VJ=15.00
MOVJ C00157 BC00157 VJ=15.00  +MOVJ EC00127 VJ=15.00
'KONIEC SZUKANIE DRUGA STRONA
'SPAWANIE DRUGA STRONA
MOVJ C00158 BC00158 VJ=15.00  +MOVJ EC00128 VJ=15.00
MACRO1 MJ#(0) ARGF7
SFTOF
SFTON P034
MOVJ C00159 BC00159 VJ=15.00  +MOVJ EC00129 VJ=15.00
ARCON
MOVL C00160 BC00160 V=10.0  +MOVJ EC00130 VJ=15.00
MOVL C00161 BC00161 V=10.0  +MOVJ EC00131 VJ=15.00
SFTOF
ARCOF
MOVJ C00162 BC00162 VJ=15.00  +MOVJ EC00132 VJ=15.00
MOVJ C00163 BC00163 VJ=50.00  +MOVJ EC00133 VJ=15.00
MOVJ C00164 BC00164 VJ=50.00  +MOVJ EC00134 VJ=50.00
MOVJ C00165 BC00165 VJ=50.00  +MOVJ EC00135 VJ=50.00
MOVJ C00166 BC00166 VJ=50.00  +MOVJ EC00136 VJ=50.00
SFTON P035
MOVL C00167 BC00167 V=83.3  +MOVJ EC00137 VJ=50.00
ARCON
MOVL C00168 BC00168 V=10.0  +MOVJ EC00138 VJ=50.00
MOVL C00169 BC00169 V=10.0  +MOVJ EC00139 VJ=50.00
ARCOF
SFTOF
MOVJ C00170 BC00170 VJ=20.00  +MOVJ EC00140 VJ=50.00
MOVJ C00171 BC00171 VJ=50.00  +MOVJ EC00141 VJ=20.00
SFTON P027
MOVJ C00172 BC00172 VJ=20.00  +MOVJ EC00142 VJ=20.00
ARCON
MOVL C00173 BC00173 V=9.2  +MOVJ EC00143 VJ=15.00
MOVL C00174 BC00174 V=9.2  +MOVJ EC00144 VJ=15.00
SFTOF
SFTON P028
MOVL C00175 BC00175 V=10.0  +MOVJ EC00145 VJ=15.00
ARCOF
MOVJ C00176 BC00176 VJ=20.00  +MOVJ EC00146 VJ=100.00
MOVJ C00177 BC00177 VJ=15.00  +MOVJ EC00147 VJ=15.00
SFTOF
MOVJ C00178 BC00178 VJ=15.00  +MOVJ EC00148 VJ=15.00
MOVJ C00179 BC00179 VJ=20.00  +MOVJ EC00149 VJ=20.00
SFTON P027
MOVJ C00180 BC00180 VJ=20.00  +MOVJ EC00150 VJ=20.00
ARCON
MOVL C00181 BC00181 V=10.0  +MOVJ EC00151 VJ=15.00
MOVL C00182 BC00182 V=10.0  +MOVJ EC00152 VJ=15.00
SFTOF
SFTON P026
MOVL C00183 BC00183 V=10.0  +MOVJ EC00153 VJ=15.00
MOVL C00184 BC00184 V=10.0  +MOVJ EC00154 VJ=15.00
ARCOF
MOVJ C00185 BC00185 VJ=15.00  +MOVJ EC00155 VJ=15.00
SFTOF
MOVJ C00186 BC00186 VJ=100.00  +MOVJ EC00156 VJ=15.00
MOVJ C00187 BC00187 VJ=100.00  +MOVJ EC00157 VJ=100.00
MOVJ C00188 BC00188 VJ=100.00  +MOVJ EC00158 VJ=100.00
MOVJ C00189 BC00189 VJ=100.00  +MOVJ EC00159 VJ=100.00
CALL JOB:CLEAN-R1_LONG
MOVJ C00190 BC00190 VJ=100.00  +MOVJ EC00160 VJ=100.00
MOVJ C00191 BC00191 VJ=100.00  +MOVJ EC00161 VJ=100.00
MOVJ C00192 BC00192 VJ=100.00  +MOVJ EC00162 VJ=100.00
MOVL C00193 BC00193 V=83.3  +MOVJ EC00163 VJ=15.00
REFP 3 RB1 C00194 BC00194
CALL JOB:SEARCH-R1
SET P021 P006
SFTON P021
MOVL C00195 BC00195 V=83.3  +MOVJ EC00164 VJ=15.00
REFP 3 RB1 C00196 BC00196
CALL JOB:SEARCH-R1
SET P021 P006
MOVL C00197 BC00197 V=83.3  +MOVJ EC00165 VJ=15.00
SFTOF
MOVL C00198 BC00198 V=166.7  +MOVJ EC00166 VJ=15.00
MOVL C00199 BC00199 V=83.3  +MOVJ EC00167 VJ=15.00
REFP 3 RB1 C00200 BC00200
CALL JOB:SEARCH-R1
SET P022 P006
SFTON P022
MOVL C00201 BC00201 V=83.3  +MOVJ EC00168 VJ=15.00
REFP 3 RB1 C00202 BC00202
CALL JOB:SEARCH-R1
SET P022 P006
MOVL C00203 BC00203 V=83.3  +MOVJ EC00169 VJ=15.00
SFTOF
MOVL C00204 BC00204 V=166.7  +MOVJ EC00170 VJ=15.00
MOVL C00205 BC00205 V=83.3  +MOVJ EC00171 VJ=15.00
REFP 3 RB1 C00206 BC00206
CALL JOB:SEARCH-R1
SET P023 P006
SFTON P023
MOVL C00207 BC00207 V=83.3  +MOVJ EC00172 VJ=15.00
REFP 3 RB1 C00208 BC00208
CALL JOB:SEARCH-R1
SET P023 P006
MOVL C00209 BC00209 V=83.3  +MOVJ EC00173 VJ=15.00
SFTOF
MOVL C00210 BC00210 V=166.7  +MOVJ EC00174 VJ=15.00
MOVL C00211 BC00211 V=83.3  +MOVJ EC00175 VJ=15.00
REFP 3 RB1 C00212 BC00212
CALL JOB:SEARCH-R1
SET P024 P006
SFTON P024
MOVL C00213 BC00213 V=83.3  +MOVJ EC00176 VJ=15.00
REFP 3 RB1 C00214 BC00214
CALL JOB:SEARCH-R1
SET P024 P006
MOVL C00215 BC00215 V=83.3  +MOVJ EC00177 VJ=15.00
SFTOF
MOVL C00216 BC00216 V=166.7  +MOVJ EC00178 VJ=15.00
MOVL C00217 BC00217 V=83.3  +MOVJ EC00179 VJ=15.00
REFP 3 RB1 C00218 BC00218
CALL JOB:SEARCH-R1
SET P025 P006
SFTON P025
MOVL C00219 BC00219 V=83.3  +MOVJ EC00180 VJ=15.00
REFP 3 RB1 C00220 BC00220
CALL JOB:SEARCH-R1
SET P025 P006
MOVL C00221 BC00221 V=133.3  +MOVJ EC00181 VJ=15.00
SFTOF
MOVJ C00222 BC00222 VJ=30.00  +MOVJ EC00182 VJ=100.00
MOVJ C00223 BC00223 VJ=30.00  +MOVJ EC00183 VJ=30.00
SFTON P023
MACRO1 MJ#(0) ARGF7
MOVL C00224 BC00224 V=83.3  +MOVJ EC00184 VJ=30.00
ARCON
SFTOF
SFTON P022
MOVL C00225 BC00225 V=10.8  +MOVJ EC00185 VJ=30.00
SFTOF
SFTON P021
MOVL C00226 BC00226 V=10.8  +MOVJ EC00186 VJ=30.00
MOVL C00227 BC00227 V=10.8  +MOVJ EC00187 VJ=30.00
ARCOF
SFTOF
MOVJ C00228 BC00228 VJ=30.00  +MOVJ EC00188 VJ=30.00
MOVJ C00229 BC00229 VJ=30.00  +MOVJ EC00189 VJ=30.00
SFTON P023
MOVL C00230 BC00230 V=83.3  +MOVJ EC00190 VJ=30.00
ARCON
SFTOF
SFTON P024
MOVL C00231 BC00231 V=10.8  +MOVJ EC00191 VJ=30.00
SFTOF
SFTON P025
MOVL C00232 BC00232 V=10.8  +MOVJ EC00192 VJ=30.00
MOVL C00233 BC00233 V=10.8  +MOVJ EC00193 VJ=30.00
MOVL C00234 BC00234 V=10.8  +MOVJ EC00194 VJ=30.00
ARCOF
SFTOF
MOVJ C00235 BC00235 VJ=30.00  +MOVJ EC00195 VJ=30.00
MOVJ C00236 BC00236 VJ=30.00  +MOVJ EC00196 VJ=30.00
MOVJ C00237 BC00237 VJ=100.00  +MOVJ EC00197 VJ=100.00
MOVJ C00238 BC00238 VJ=30.00  +MOVJ EC00198 VJ=30.00
CALL JOB:ONLYCUT-R1_LONG
MOVJ C00239 BC00239 VJ=30.00  +MOVJ EC00199 VJ=30.00
MOVJ C00240 BC00240 VJ=100.00  +MOVJ EC00200 VJ=100.00
MOVJ C00241 BC00241 VJ=60.00  +MOVJ EC00201 VJ=30.00
MOVJ C00242 BC00242 VJ=60.00  +MOVJ EC00202 VJ=30.00
MOVJ C00243 BC00243 VJ=60.00  +MOVJ EC00203 VJ=30.00
MOVJ C00244 BC00244 VJ=60.00  +MOVJ EC00204 VJ=30.00
MOVJ C00245 BC00245 VJ=100.00  +MOVJ EC00205 VJ=100.00
MOVL C00246 BC00246 V=83.3  +MOVJ EC00206 VJ=15.00
REFP 3 RB1 C00247 BC00247
CALL JOB:SEARCH-R1
SET P021 P006
SFTON P021
MOVL C00248 BC00248 V=83.3  +MOVJ EC00207 VJ=15.00
REFP 3 RB1 C00249 BC00249
CALL JOB:SEARCH-R1
SET P021 P006
MOVL C00250 BC00250 V=83.3  +MOVJ EC00208 VJ=15.00
SFTOF
MOVL C00251 BC00251 V=166.7  +MOVJ EC00209 VJ=15.00
MOVL C00252 BC00252 V=83.3  +MOVJ EC00210 VJ=15.00
REFP 3 RB1 C00253 BC00253
CALL JOB:SEARCH-R1
SET P022 P006
SFTON P022
MOVL C00254 BC00254 V=83.3  +MOVJ EC00211 VJ=15.00
REFP 3 RB1 C00255 BC00255
CALL JOB:SEARCH-R1
SET P022 P006
MOVL C00256 BC00256 V=83.3  +MOVJ EC00212 VJ=15.00
SFTOF
MOVL C00257 BC00257 V=166.7  +MOVJ EC00213 VJ=15.00
MOVL C00258 BC00258 V=83.3  +MOVJ EC00214 VJ=15.00
REFP 3 RB1 C00259 BC00259
CALL JOB:SEARCH-R1
SET P023 P006
SFTON P023
MOVL C00260 BC00260 V=83.3  +MOVJ EC00215 VJ=15.00
REFP 3 RB1 C00261 BC00261
CALL JOB:SEARCH-R1
SET P023 P006
MOVL C00262 BC00262 V=83.3  +MOVJ EC00216 VJ=15.00
SFTOF
MOVL C00263 BC00263 V=166.7  +MOVJ EC00217 VJ=15.00
MOVL C00264 BC00264 V=83.3  +MOVJ EC00218 VJ=15.00
REFP 3 RB1 C00265 BC00265
CALL JOB:SEARCH-R1
SET P024 P006
SFTON P024
MOVL C00266 BC00266 V=83.3  +MOVJ EC00219 VJ=15.00
REFP 3 RB1 C00267 BC00267
CALL JOB:SEARCH-R1
SET P024 P006
MOVL C00268 BC00268 V=83.3  +MOVJ EC00220 VJ=15.00
SFTOF
MOVL C00269 BC00269 V=166.7  +MOVJ EC00221 VJ=15.00
MOVL C00270 BC00270 V=83.3  +MOVJ EC00222 VJ=15.00
REFP 3 RB1 C00271 BC00271
CALL JOB:SEARCH-R1
SET P025 P006
SFTON P025
MOVL C00272 BC00272 V=83.3  +MOVJ EC00223 VJ=15.00
REFP 3 RB1 C00273 BC00273
CALL JOB:SEARCH-R1
SET P025 P006
MOVL C00274 BC00274 V=83.3  +MOVJ EC00224 VJ=15.00
SFTOF
MOVJ C00275 BC00275 VJ=30.00  +MOVJ EC00225 VJ=100.00
MOVJ C00276 BC00276 VJ=30.00  +MOVJ EC00226 VJ=30.00
SFTON P023
MOVL C00277 BC00277 V=83.3  +MOVJ EC00227 VJ=30.00
ARCON
SFTOF
SFTON P022
MOVL C00278 BC00278 V=10.8  +MOVJ EC00228 VJ=30.00
SFTOF
SFTON P021
MOVL C00279 BC00279 V=10.8  +MOVJ EC00229 VJ=30.00
MOVL C00280 BC00280 V=10.8  +MOVJ EC00230 VJ=30.00
ARCOF
SFTOF
MOVJ C00281 BC00281 VJ=30.00  +MOVJ EC00231 VJ=30.00
MOVJ C00282 BC00282 VJ=30.00  +MOVJ EC00232 VJ=30.00
SFTON P023
MOVL C00283 BC00283 V=83.3  +MOVJ EC00233 VJ=30.00
ARCON
SFTOF
SFTON P024
MOVL C00284 BC00284 V=10.8  +MOVJ EC00234 VJ=30.00
SFTOF
SFTON P025
MOVL C00285 BC00285 V=10.8  +MOVJ EC00235 VJ=30.00
MOVL C00286 BC00286 V=10.8  +MOVJ EC00236 VJ=30.00
MOVL C00287 BC00287 V=10.8  +MOVJ EC00237 VJ=30.00
ARCOF
SFTOF
MOVJ C00288 BC00288 VJ=50.00  +MOVJ EC00238 VJ=30.00
MOVJ C00289 BC00289 VJ=50.00  +MOVJ EC00239 VJ=30.00
MOVJ C00290 BC00290 VJ=50.00  +MOVJ EC00240 VJ=30.00
MOVJ C00291 BC00291 VJ=100.00  +MOVJ EC00241 VJ=100.00
PAUSE
PAUSE
'ZALOZYC USZY ZE SCIANY
MOVJ C00292 BC00292 VJ=100.00  +MOVJ EC00242 VJ=100.00
END
